// TIA Portal V20 export
// export: Created 2025-09-14T10:59:00.0000000Z, ExportSetting WithDefaults
VAR_GLOBAL   // PLC tag table "TagTable_DI"
   RTU1_SF_RunFdbk AT %I0.0 : Bool;
   RTU1_SF_AirflowSw AT %I0.1 : Bool;
   RTU1_SF_VfdFault AT %I0.2 : Bool;
   RTU1_C_HighPressSw AT %I0.3 : Bool;
   RTU1_C_LowPressSw AT %I0.4 : Bool;
   RTU1_C_FreezeStat AT %I0.5 : Bool;
   RTU1_H_HighTempSw AT %I0.6 : Bool;
   RTU1_SYS_DirtyFilter AT %I0.7 : Bool;
END_VAR
